// Mitsubishi GX Works2 project: FX1s_encoderAB   PLC: FX1S

PROGRAM MAIN
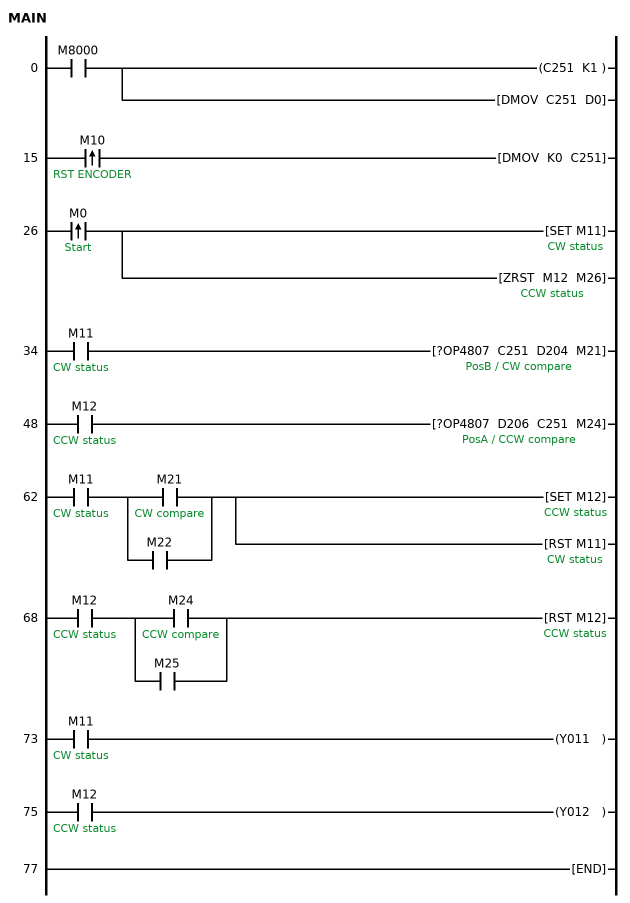
0     LD      M8000
      OUT     C251 K1
      DMOV    C251 D0
15    LDP     M10  ; RST ENCODER
      DMOV    K0 C251
26    LDP     M0  ; Start
      SET     M11  ; CW status
      ZRST    M12 M26  ; CCW status
34    LD      M11  ; CW status
      ?OP4807 C251 D204 M21  ; PosB / CW compare
48    LD      M12  ; CCW status
      ?OP4807 D206 C251 M24  ; PosA / CCW compare
62    LD      M11  ; CW status
      LD      M21  ; CW compare
      OR      M22
      ANB
      SET     M12  ; CCW status
      RST     M11  ; CW status
68    LD      M12  ; CCW status
      LD      M24  ; CCW compare
      OR      M25
      ANB
      RST     M12  ; CCW status
73    LD      M11  ; CW status
      OUT     Y011
75    LD      M12  ; CCW status
      OUT     Y012
77    END
END_PROGRAM
